(* IEC 61131-3 sources: ATCMcontrol_Engineering/src/COM/softing/fc/AddOns/Softing/4CPCTarget/Libs/ATCM_FLib, 23 files *)

(* ---- FA_SYNC_CLOSEFILE.st ---- *)
(*[[
    UserURL= "ATCM:FA_SYNC_CLOSEFILE.htm"
]]*)

(*
 *  ATCMControl FileAccess Function FA_SYNC_CLOSEFILE
 *  Purpose: Closes a file after read, write or getsize operation.
 *)
FUNCTION FA_SYNC_CLOSEFILE:BOOL     (* Return Value: error flag *)
VAR_INPUT
    EXEC        : BOOL;             (* start operation *)
END_VAR
VAR_IN_OUT
    FILE        : FA_SYNC_FILE;     (* file instance to operate on *)
END_VAR

inline
{
    ((COM.softing.fclib.flib.SyncFLib)%2).closeFile(%1)
}
END_FUNCTION

(* ---- FA_SYNC_CREATEDIRECTORY.st ---- *)
(*[[
    UserURL= "ATCM:FA_SYNC_CREATEDIRECTORY.htm"
]]*)

(*
 *  ATCMControl FileAccess Function FA_SYNC_CREATEDIRECTORY
 *  Purpose: Create a new directory.
 *)
FUNCTION FA_SYNC_CREATEDIRECTORY:BOOL   (* Return Value: error flag *)
VAR_INPUT
    EXEC        : BOOL;                 (* start operation *)
END_VAR
VAR_IN_OUT
    FILE        : FA_SYNC_FILE;         (* file instance to operate on *)
END_VAR

inline
{
    ((COM.softing.fclib.flib.SyncFLib)%2).createDir(%1)
}
END_FUNCTION

(* ---- FA_SYNC_DELETEFILE.st ---- *)
(*[[
    UserURL= "ATCM:FA_SYNC_DELETEFILE.htm"
]]*)

(*
 *  ATCMControl FileAccess Function FA_SYNC_DELETEFILE
 *  Purpose: Delete a file.
 *)
FUNCTION FA_SYNC_DELETEFILE:BOOL    (* Return Value: error flag *)
VAR_INPUT
    EXEC        : BOOL;             (* start operation *)
END_VAR
VAR_IN_OUT
    FILE        : FA_SYNC_FILE;     (* file instance to operate on *)
END_VAR

inline
{
    ((COM.softing.fclib.flib.SyncFLib)%2).deleteFile(%1)
}
END_FUNCTION

(* ---- FA_SYNC_EXISTSFILE.st ---- *)
(*[[
    UserURL= "ATCM:FA_SYNC_EXISTSFILE.htm"
]]*)

(*
 *  ATCMControl FileAccess Function FA_SYNC_EXISTSFILE
 *  Purpose: Determines whether a file exists.
 *)
FUNCTION FA_SYNC_EXISTSFILE:BOOL    (* Return Value: error flag *)
VAR_INPUT
    EXEC        : BOOL;             (* start operation *)
END_VAR
VAR_IN_OUT
    FILE        : FA_SYNC_FILE;     (* file instance to operate on *)
END_VAR
VAR_OUTPUT
    EXISTS      : BOOL;             (* TRUE if files exists, else FALSE *)
END_VAR

inline
{
    ((COM.softing.fclib.flib.SyncFLib)%2).existsFile(%1, %3)
}
END_FUNCTION

(* ---- FA_SYNC_GETSIZE.st ---- *)
(*[[
    UserURL= "ATCM:FA_SYNC_GETSIZE.htm"
]]*)

(*
 *  ATCMControl FileAccess Function FA_SYNC_GETSIZE
 *  Purpose: Retrieves the length in bytes of a file.
 *)
FUNCTION FA_SYNC_GETSIZE:BOOL       (* Return Value: error flag *)
VAR_INPUT
    EXEC        : BOOL;             (* start operation *)
END_VAR
VAR_IN_OUT
    FILE        : FA_SYNC_FILE;     (* file instance to operate on *)
END_VAR
VAR_OUTPUT
    SIZE        : LINT;             (* file size in bytes *)
END_VAR

inline
{
    ((COM.softing.fclib.flib.SyncFLib)%2).getSize(%1, %3)
}
END_FUNCTION

(* ---- FA_SYNC_OPENFILE.st ---- *)
(*[[
    UserURL= "ATCM:FA_SYNC_OPENFILE.htm"
]]*)

(*
 *  ATCMControl FileAccess Function FA_SYNC_OPENFILE
 *  Purpose: Opens a file for read, write or getsize operations.
 *)
FUNCTION FA_SYNC_OPENFILE:BOOL      (* Return Value: error flag *)
VAR_INPUT
    EXEC        : BOOL;             (* start operation *)
END_VAR
VAR_IN_OUT
    FILE        : FA_SYNC_FILE;     (* file instance to operate on *)
END_VAR

inline
{
    ((COM.softing.fclib.flib.SyncFLib)%2).createFile(%1)
}
END_FUNCTION

(* ---- FA_SYNC_READFILE.st ---- *)
(*[[
    UserURL= "ATCM:FA_SYNC_READFILE.htm"
]]*)

(*
 *  ATCMControl FileAccess Function FA_SYNC_READFILE
 *  Purpose: Reads data from a file.
 *)
FUNCTION FA_SYNC_READFILE:BOOL      (* Return Value: error flag *)
VAR_INPUT
    EXEC        : BOOL;             (* start operation *)
END_VAR
VAR_IN_OUT
    FILE        : FA_SYNC_FILE;     (* file instance to operate on *)
    LENGTH      : DINT;             (* bytes to read; return read bytes *)
END_VAR
VAR_OUTPUT
    DATA        : BYTE_STRING;      (* read data *)
END_VAR

inline
{
    ((COM.softing.fclib.flib.SyncFLib)%2).readFile(%1, %3, %4)
}
END_FUNCTION

(* ---- FA_SYNC_RENAMEFILE.st ---- *)
(*[[
    UserURL= "ATCM:FA_SYNC_RENAMEFILE.htm"
]]*)

(*
 *  ATCMControl FileAccess Function FA_SYNC_RENAMEFILE
 *  Purpose: Close file after read, write or getsize operation.
 *)
FUNCTION FA_SYNC_RENAMEFILE:BOOL    (* Return Value: error flag *)
VAR_INPUT
    EXEC        : BOOL;             (* start operation *)
    NEWNAME     : WSTRING;          (* new filename *)
END_VAR
VAR_IN_OUT
    FILE        : FA_SYNC_FILE;     (* file instance to operate on *)
END_VAR

inline
{
    ((COM.softing.fclib.flib.SyncFLib)%3).renameFile(%1, %2)
}
END_FUNCTION

(* ---- FA_SYNC_WRITEFILE.st ---- *)
(*[[
    UserURL= "ATCM:FA_SYNC_WRITEFILE.htm"
]]*)

(*
 *  ATCMControl FileAccess Function FA_SYNC_WRITEFILE
 *  Purpose: Writes data to a file.
 *)
FUNCTION FA_SYNC_WRITEFILE:BOOL     (* Return Value: error flag *)
VAR_INPUT
    EXEC        : BOOL;             (* start operation *)
    DATA        : BYTE_STRING;      (* data to write *)
END_VAR
VAR_IN_OUT
    FILE        : FA_SYNC_FILE;     (* file instance to operate on *)
END_VAR

inline
{
    ((COM.softing.fclib.flib.SyncFLib)%3).writeFile(%1, %2)
}
END_FUNCTION

(* ---- FA_ASYNC_CLOSEFILE.st ---- *)
(*[[
    UserURL= "ATCM:FA_ASYNC_CLOSEFILE.htm"
]]*)

(*
 *  ATCMControl FileAccess Functionblock FA_ASYNC_CLOSEFILE
 *  Purpose: Closes a file after read, write or getsize operation.
 *)
FUNCTION_BLOCK FA_ASYNC_CLOSEFILE
VAR_INPUT
    EXEC        : BOOL;             (* raising edge starts operation *)
END_VAR
VAR_IN_OUT
    FILE        : FA_ASYNC_FILE;    (* file instance to operate on *)
END_VAR
VAR_OUTPUT
    DONE        : BOOL;             (* operation finished *)
    ERROR       : BOOL;             (* error flag *)
    ERRCD       : DINT;             (* error code *)
    ERRTXT      : WSTRING;          (* error text *)
END_VAR

VAR
    rtrigExec   : R_TRIG;           (* execute *)
    token       : BOOL;             (* instance access token *)
    ireq        : BOOL;             (* execute request *)
END_VAR

rtrigExec(CLK := EXEC);
ireq := rtrigExec.Q;

NATIVE
    _done.putBool( ((COM.softing.fclib.flib.AsyncFLib)_file).closeFile(_exec.getBool(),
                        _ireq.getBool(),
                        _token,
                        this,
                        _error,
                        _errcd,
                        _errtxt) );
END_NATIVE;

END_FUNCTION_BLOCK

(* ---- FA_ASYNC_COPYFILE.st ---- *)
(*[[
    UserURL= "ATCM:FA_ASYNC_COPYFILE.htm"
]]*)

(*
 *  ATCMControl FileAccess Functionblock FA_ASYNC_COPYFILE
 *  Purpose: Copy a file.
 *)
FUNCTION_BLOCK FA_ASYNC_COPYFILE

VAR_INPUT
    EXEC        : BOOL;             (* raising edge starts operation *)
    DESTNAME    : WSTRING;          (* destination filename *)
    OVERWRITE   : BOOL := TRUE;     (* enable overwrite mode *)
END_VAR
VAR_IN_OUT
    FILE        : FA_ASYNC_FILE;    (* file instance to operate on *)
END_VAR
VAR_OUTPUT
    DONE        : BOOL;             (* operation finished *)
    ERROR       : BOOL;             (* error flag *)
    ERRCD       : DINT;             (* error code *)
    ERRTXT      : WSTRING;          (* error text *)
END_VAR

VAR
    rtrigExec   : R_TRIG;           (* execute *)
    token       : BOOL;             (* instance access token *)
    ireq        : BOOL;             (* execute request *)
END_VAR

rtrigExec(CLK := EXEC);
ireq := rtrigExec.Q;

NATIVE
    _done.putBool( ((COM.softing.fclib.flib.AsyncFLib)_file).copyFile(_exec.getBool(),
                        _ireq.getBool(),
                        _token,
                        this,
                        _destname.getString(),
                        _overwrite.getBool(),
                        _error,
                        _errcd,
                        _errtxt) );
END_NATIVE;

END_FUNCTION_BLOCK

(* ---- FA_ASYNC_CREATEDIRECTORY.st ---- *)
(*[[
    UserURL= "ATCM:FA_ASYNC_CREATEDIRECTORY.htm"
]]*)

(*
 *  ATCMControl FileAccess Functionblock FA_ASYNC_CREATEDIRECTORY
 *  Purpose: Create a new directory.
 *)
FUNCTION_BLOCK FA_ASYNC_CREATEDIRECTORY
VAR_INPUT
    EXEC        : BOOL;             (* raising edge starts operation *)
END_VAR
VAR_IN_OUT
    FILE        : FA_ASYNC_FILE;    (* file instance to operate on *)
END_VAR
VAR_OUTPUT
    DONE        : BOOL;             (* operation finished *)
    ERROR       : BOOL;             (* error flag *)
    ERRCD       : DINT;             (* error code *)
    ERRTXT      : WSTRING;          (* error text *)
END_VAR

VAR
    rtrigExec   : R_TRIG;           (* execute *)
    token       : BOOL;             (* instance access token *)
    ireq        : BOOL;             (* execute request *)
END_VAR

rtrigExec(CLK := EXEC);
ireq := rtrigExec.Q;

NATIVE
    _done.putBool( ((COM.softing.fclib.flib.AsyncFLib)_file).createDir(_exec.getBool(),
                        _ireq.getBool(),
                        _token,
                        this,
                        _error,
                        _errcd,
                        _errtxt) );
END_NATIVE;

END_FUNCTION_BLOCK

(* ---- FA_ASYNC_DELETEFILE.st ---- *)
(*[[
    UserURL= "ATCM:FA_ASYNC_DELETEFILE.htm"
]]*)

(*
 *  ATCMControl FileAccess Functionblock FA_ASYNC_DELETEFILE
 *  Purpose: Delete a file.
 *)
FUNCTION_BLOCK FA_ASYNC_DELETEFILE
VAR_INPUT
    EXEC        : BOOL;             (* raising edge starts operation *)
END_VAR
VAR_IN_OUT
    FILE        : FA_ASYNC_FILE;    (* file instance to operate on *)
END_VAR
VAR_OUTPUT
    DONE        : BOOL;             (* operation finished *)
    ERROR       : BOOL;             (* error flag *)
    ERRCD       : DINT;             (* error code *)
    ERRTXT      : WSTRING;          (* error text *)
END_VAR

VAR
    rtrigExec   : R_TRIG;           (* execute *)
    token       : BOOL;             (* instance access token *)
    ireq        : BOOL;             (* execute request *)
END_VAR

rtrigExec(CLK := EXEC);
ireq := rtrigExec.Q;

NATIVE
    _done.putBool( ((COM.softing.fclib.flib.AsyncFLib)_file).deleteFile(_exec.getBool(),
                        _ireq.getBool(),
                        _token,
                        this,
                        _error,
                        _errcd,
                        _errtxt) );
END_NATIVE;

END_FUNCTION_BLOCK

(* ---- FA_ASYNC_EXISTSFILE.st ---- *)
(*[[
    UserURL= "ATCM:FA_ASYNC_EXISTSFILE.htm"
]]*)

(*
 *  ATCMControl FileAccess Functionblock FA_ASYNC_EXISTSFILE
 *  Purpose: Determines whether a file exists.
 *)
FUNCTION_BLOCK FA_ASYNC_EXISTSFILE
VAR_INPUT
    EXEC        : BOOL;             (* raising edge starts operation *)
END_VAR
VAR_IN_OUT
    FILE        : FA_ASYNC_FILE;    (* file instance to operate on *)
END_VAR
VAR_OUTPUT
    EXISTS      : BOOL;             (* TRUE if files exists, else FALSE *)
    DONE        : BOOL;             (* operation finished *)
    ERROR       : BOOL;             (* error flag *)
    ERRCD       : DINT;             (* error code *)
    ERRTXT      : WSTRING;          (* error text *)
END_VAR

VAR
    rtrigExec   : R_TRIG;           (* execute *)
    token       : BOOL;             (* instance access token *)
    ireq        : BOOL;             (* execute request *)
END_VAR

rtrigExec(CLK := EXEC);
ireq := rtrigExec.Q;

NATIVE
    _done.putBool( ((COM.softing.fclib.flib.AsyncFLib)_file).existsFile(_exec.getBool(),
                        _ireq.getBool(),
                        _token,
                        this,
                        _exists,
                        _error,
                        _errcd,
                        _errtxt) );
END_NATIVE;

END_FUNCTION_BLOCK

(* ---- FA_ASYNC_GETSIZE.st ---- *)
(*[[
    UserURL= "ATCM:FA_ASYNC_GETSIZE.htm"
]]*)

(*
 *  ATCMControl FileAccess Functionblock FA_ASYNC_GETSIZE
 *  Purpose: Retrieves the length in bytes of a file.
 *)
FUNCTION_BLOCK FA_ASYNC_GETSIZE
VAR_INPUT
    EXEC        : BOOL;             (* raising edge starts operation *)
END_VAR
VAR_IN_OUT
    FILE        : FA_ASYNC_FILE;    (* file instance to operate on *)
END_VAR
VAR_OUTPUT
    SIZE        : LINT;             (* file size in bytes *)
    DONE        : BOOL;             (* operation finished *)
    ERROR       : BOOL;             (* error flag *)
    ERRCD       : DINT;             (* error code *)
    ERRTXT      : WSTRING;          (* error text *)
END_VAR

VAR
    rtrigExec   : R_TRIG;           (* execute *)
    token       : BOOL;             (* instance access token *)
    ireq        : BOOL;             (* execute request *)
END_VAR

rtrigExec(CLK := EXEC);
ireq := rtrigExec.Q;

NATIVE
    _done.putBool( ((COM.softing.fclib.flib.AsyncFLib)_file).getSize(_exec.getBool(),
                        _ireq.getBool(),
                        _token,
                        this,
                        (FcObject)_size,
                        _error,
                        _errcd,
                        _errtxt) );
END_NATIVE;

END_FUNCTION_BLOCK

(* ---- FA_ASYNC_OPENFILE.st ---- *)
(*[[
    UserURL= "ATCM:FA_ASYNC_OPENFILE.htm"
]]*)

(*
 *  ATCMControl FileAccess Functionblock FA_ASYNC_OPENFILE
 *  Purpose: Opens a file for read, write or getsize operations.
 *)
FUNCTION_BLOCK FA_ASYNC_OPENFILE
VAR_INPUT
    EXEC        : BOOL;             (* raising edge starts operation *)
END_VAR
VAR_IN_OUT
    FILE        : FA_ASYNC_FILE;    (* file instance to operate on *)
END_VAR
VAR_OUTPUT
    DONE        : BOOL;             (* operation finished *)
    ERROR       : BOOL;             (* error flag *)
    ERRCD       : DINT;             (* error code *)
    ERRTXT      : WSTRING;          (* error text *)
END_VAR

VAR
    rtrigExec   : R_TRIG;           (* execute *)
    token       : BOOL;             (* instance access token *)
    ireq        : BOOL;             (* execute request *)
END_VAR

rtrigExec(CLK := EXEC);
ireq := rtrigExec.Q;

NATIVE
    _done.putBool( ((COM.softing.fclib.flib.AsyncFLib)_file).createFile(_exec.getBool(),
                        _ireq.getBool(),
                        _token,
                        this,
                        _error,
                        _errcd,
                        _errtxt) );
END_NATIVE;

END_FUNCTION_BLOCK

(* ---- FA_ASYNC_READFILE.st ---- *)
(*[[
    UserURL= "ATCM:FA_ASYNC_READFILE.htm"
]]*)

(*
 *  ATCMControl FileAccess Functionblock FA_ASYNC_READFILE
 *  Purpose: Reads data from a file.
 *)

FUNCTION_BLOCK FA_ASYNC_READFILE
VAR_INPUT
    EXEC        : BOOL;             (* raising edge starts operation *)
END_VAR
VAR_IN_OUT
    FILE        : FA_ASYNC_FILE;    (* file instance to operate on *)
    LENGTH      : DINT;             (* bytes to read; return read bytes *)
END_VAR
VAR_OUTPUT
    DATA        : BYTE_STRING;      (* read data *)
    DONE        : BOOL;             (* operation finished *)
    ERROR       : BOOL;             (* error flag *)
    ERRCD       : DINT;             (* error code *)
    ERRTXT      : WSTRING;          (* error text *)
END_VAR

VAR
    rtrigExec   : R_TRIG;           (* execute *)
    token       : BOOL;             (* instance access token *)
    ireq        : BOOL;             (* execute request *)
END_VAR

rtrigExec(CLK := EXEC);
ireq := rtrigExec.Q;

NATIVE
    _done.putBool( ((COM.softing.fclib.flib.AsyncFLib)_file).readFile(_exec.getBool(),
                        _ireq.getBool(),
                        _token,
                        this,
                        (FcObject)_data,
                        _length,
                        _error,
                        _errcd,
                        _errtxt) );
END_NATIVE;

END_FUNCTION_BLOCK

(* ---- FA_ASYNC_RENAMEFILE.st ---- *)
(*[[
    UserURL= "ATCM:FA_ASYNC_RENAMEFILE.htm"
]]*)

(*
 *  ATCMControl FileAccess Functionblock FA_ASYNC_RENAMEFILE
 *  Purpose: Close file after read, write or getsize operation.
 *)
FUNCTION_BLOCK FA_ASYNC_RENAMEFILE
VAR_INPUT
    EXEC        : BOOL;             (* raising edge starts operation *)
    NEWNAME     : WSTRING;          (* new filename *)
END_VAR
VAR_IN_OUT
    FILE        : FA_ASYNC_FILE;    (* file instance to operate on *)
END_VAR
VAR_OUTPUT
    DONE        : BOOL;             (* operation finished *)
    ERROR       : BOOL;             (* error flag *)
    ERRCD       : DINT;             (* error code *)
    ERRTXT      : WSTRING;          (* error text *)
END_VAR

VAR
    rtrigExec   : R_TRIG;           (* execute *)
    token       : BOOL;             (* instance access token *)
    ireq        : BOOL;             (* execute request *)
END_VAR

rtrigExec(CLK := EXEC);
ireq := rtrigExec.Q;

NATIVE
    _done.putBool( ((COM.softing.fclib.flib.AsyncFLib)_file).renameFile(_exec.getBool(),
                        _ireq.getBool(),
                        _token,
                        this,
                        _newname.getString(),
                        _error,
                        _errcd,
                        _errtxt) );
END_NATIVE;

END_FUNCTION_BLOCK

(* ---- FA_ASYNC_WRITEFILE.st ---- *)
(*[[
    UserURL= "ATCM:FA_ASYNC_WRITEFILE.htm"
]]*)

(*
 *  ATCMControl FileAccess Functionblock FA_ASYNC_WRITEFILE
 *  Purpose: Writes data to a file.
 *)
FUNCTION_BLOCK FA_ASYNC_WRITEFILE
VAR_INPUT
    EXEC        : BOOL;             (* raising edge starts operation *)
    DATA        : BYTE_STRING;      (* data to write *)
END_VAR
VAR_IN_OUT
    FILE        : FA_ASYNC_FILE;    (* file instance to operate on *)
END_VAR
VAR_OUTPUT
    DONE        : BOOL;             (* operation finished *)
    ERROR       : BOOL;             (* error flag *)
    ERRCD       : DINT;             (* error code *)
    ERRTXT      : WSTRING;          (* error text *)
END_VAR

VAR
    rtrigExec   : R_TRIG;           (* execute *)
    token       : BOOL;             (* instance access token *)
    ireq        : BOOL;             (* execute request *)
END_VAR

rtrigExec(CLK := EXEC);
ireq := rtrigExec.Q;

NATIVE
    _done.putBool( ((COM.softing.fclib.flib.AsyncFLib)_file).writeFile(_exec.getBool(),
                        _ireq.getBool(),
                        _token,
                        this,
                        _data,
                        _error,
                        _errcd,
                        _errtxt) );
END_NATIVE;

END_FUNCTION_BLOCK

(* ---- FA_READFILE.st ---- *)
(*[[
    UserURL= "ATCM:FA_READFILE.htm"
]]*)

(*
 *  ATCMControl FileAccess Functionblock FA_READFILE
 *  Purpose: Reads data from a file.
 *)
FUNCTION_BLOCK FA_READFILE
VAR_INPUT
    EXEC        : BOOL;             (* raising edge starts operation *)
    FILENAME    : WSTRING;          (* filename *)
    TOUT        : TIME;             (* timeout for this operation *)
END_VAR
VAR_IN_OUT
    POSITION    : DINT;             (* start at position; returns last position *)
    LENGTH      : DINT;             (* bytes to read; returns read bytes *)
END_VAR
VAR_OUTPUT
    DATA        : BYTE_STRING;      (* read data *)
    DONE        : BOOL;             (* operation finished *)
    ERROR       : BOOL;             (* error flag *)
    ERRCD       : DINT;             (* error code *)
    ERRTXT      : WSTRING;          (* error text *)
END_VAR

VAR
    file        : FA_ASYNC_FILE;
    aopen       : FA_ASYNC_OPENFILE;
    aread       : FA_ASYNC_READFILE;
    aclose      : FA_ASYNC_CLOSEFILE;
    rtDone      : R_TRIG;
    rtInit      : R_TRIG;
    rtRead      : R_TRIG;
    rtError     : R_TRIG;
    bstrData    : BYTE_STRING;
END_VAR

(* init structure *)
file.FILENAME := FILENAME;
file.MODE := CFA_READ;
(* file.TEXTMODE is default: FALSE *)
file.TOUT := TOUT;

(* delete output *)
IF NOT EXEC THEN
    DONE := FALSE;
    ERROR := FALSE;
    ERRCD := 0;
    ERRTXT := "";
    BYTE_STRING_INIT(DATA, "");
    file.ISERROR := FALSE;
END_IF;

(* open file *)
aopen(EXEC := EXEC, FILE := file);

(* init read file *)
rtInit(CLK := aopen.DONE);
IF rtInit.Q THEN
    (* init *)
    file.POSITION := POSITION;
END_IF;
aread(EXEC := aopen.DONE AND NOT aopen.ERROR, FILE := file, LENGTH := LENGTH);
(* read file done *)
rtRead(CLK := aread.DONE);
IF rtRead.Q THEN
    bstrData := aread.DATA;
END_IF;

(* close file *)
aclose(EXEC := aread.DONE AND NOT aread.ERROR, FILE := file);

(* init output vars *)
rtDone(CLK := aclose.DONE);
IF rtDone.Q THEN
    DONE        := TRUE;
    DATA        := bstrData;
    POSITION    := file.POSITION;
END_IF;

(* init error vars *)
rtError(CLK := file.ISERROR);
IF rtError.Q THEN
    DONE        := TRUE;
    BYTE_STRING_INIT(DATA, "");
    ERROR       := file.ISERROR;
    ERRCD       := file.LSTERRCD;
    ERRTXT      := file.LSTERRTXT;
END_IF;

END_FUNCTION_BLOCK

(* ---- FA_READLINE.st ---- *)
(*[[
    UserURL= "ATCM:FA_READLINE.htm"
]]*)

(*
 *  ATCMControl FileAccess Functionblock FA_READLINE
 *  Purpose: Reads data from a file.
 *)
FUNCTION_BLOCK FA_READLINE
VAR_INPUT
    EXEC        : BOOL;             (* raising edge starts operation *)
    FILENAME    : WSTRING;          (* filename *)
    TOUT        : TIME;             (* timeout for this operation *)
END_VAR
VAR_IN_OUT
    POSITION    : DINT;             (* start at position; returns last position *)
END_VAR
VAR_OUTPUT
    DATA        : WSTRING;          (* read data *)
    DONE        : BOOL;             (* operation finished *)
    ERROR       : BOOL;             (* error flag *)
    ERRCD       : DINT;             (* error code *)
    ERRTXT      : WSTRING;          (* error text *)
END_VAR

VAR
    file        : FA_ASYNC_FILE;
    aopen       : FA_ASYNC_OPENFILE;
    aread       : FA_ASYNC_READFILE;
    aclose      : FA_ASYNC_CLOSEFILE;
    length      : DINT;
    rtDone      : R_TRIG;
    rtInit      : R_TRIG;
    rtRead      : R_TRIG;
    rtError     : R_TRIG;
    pos         : DINT;
    bstrData    : BYTE_STRING;
END_VAR

(* init structure *)
file.FILENAME := FILENAME;
file.MODE := CFA_READ;
file.TEXTMODE := TRUE;
file.TOUT := TOUT;
length := CFA_EOL;

(* delete output *)
IF NOT EXEC THEN
    DONE := FALSE;
    ERROR := FALSE;
    ERRCD := 0;
    ERRTXT := "";
    DATA := "";
    file.ISERROR := FALSE;
END_IF;

(* open file *)
aopen(EXEC := EXEC, FILE := file);

(* init read file *)
rtInit(CLK := aopen.DONE);
IF rtInit.Q THEN
    (* init *)
    file.POSITION := POSITION;
END_IF;
aread(EXEC := aopen.DONE AND NOT aopen.ERROR, FILE := file, LENGTH := length);
(* read file done *)
rtRead(CLK := aread.DONE);
IF rtRead.Q THEN
    bstrData := aread.DATA;
END_IF;

(* close file *)
aclose(EXEC := aread.DONE AND NOT aread.ERROR, FILE := file);

(* init output vars *)
rtDone(CLK := aclose.DONE);
IF rtDone.Q THEN
    DONE        := TRUE;
    (* convert WString to BYTE_STRING *)
    pos := 0;
    DATA        := COPY_WSTRING_FROM_BYTE_STRING(bstrdata.SIZE, pos, bstrdata);
    POSITION    := file.POSITION;
END_IF;

(* init error vars *)
rtError(CLK := file.ISERROR);
IF rtError.Q THEN
    DONE        := TRUE;
    DATA        := "";
    ERROR       := file.ISERROR;
    ERRCD       := file.LSTERRCD;
    ERRTXT      := file.LSTERRTXT;
END_IF;

END_FUNCTION_BLOCK

(* ---- FA_WRITEFILE.st ---- *)
(*[[
    UserURL= "ATCM:FA_WRITEFILE.htm"
]]*)

(*
 *  ATCMControl FileAccess Functionblock FA_WRITEFILE
 *  Purpose: Writes data to a file.
 *)
FUNCTION_BLOCK FA_WRITEFILE
VAR_INPUT
    EXEC        : BOOL;             (* raising edge starts operation *)
    FILENAME    : WSTRING;          (* filename *)
    TOUT        : TIME;             (* timeout for this operation *)
    DATA        : BYTE_STRING;      (* data to write *)
END_VAR
VAR_IN_OUT
    POSITION    : DINT;             (* start at position; returns last position *)
END_VAR
VAR_OUTPUT
    DONE        : BOOL;             (* operation finished *)
    ERROR       : BOOL;             (* error flag *)
    ERRCD       : DINT;             (* error code *)
    ERRTXT      : WSTRING;          (* error text *)
END_VAR

VAR
    file        : FA_ASYNC_FILE;
    aopen       : FA_ASYNC_OPENFILE;
    awrite      : FA_ASYNC_WRITEFILE;
    aclose      : FA_ASYNC_CLOSEFILE;
    rtWrite     : R_TRIG;
    rtDone      : R_TRIG;
    rtError     : R_TRIG;
    posPtr      : DINT;
END_VAR

(* init structure *)
file.FILENAME := FILENAME;
file.MODE := CFA_READ_WRITE;
(* file.TEXTMODE is default: FALSE *)
file.TOUT := TOUT;

(* delete output *)
IF NOT EXEC THEN
    DONE := FALSE;
    ERROR := FALSE;
    ERRCD := 0;
    ERRTXT := "";
    file.ISERROR := FALSE;
END_IF;

(* open file *)
aopen(EXEC := EXEC, FILE := file);

(* read file *)
file.POSITION := POSITION;
awrite(EXEC := aopen.DONE AND NOT aopen.ERROR, FILE := file, DATA := DATA);
(* write file done *)
rtWrite(CLK := awrite.DONE);
IF rtWrite.Q THEN
    posPtr := file.POSITION;
END_IF;

(* close file *)
aclose(EXEC := awrite.DONE, FILE := file);

(* init output vars *)
rtDone(CLK := aclose.DONE);
IF rtDone.Q THEN
    DONE        := TRUE;
    POSITION    := posPtr;
END_IF;

(* init error vars *)
rtError(CLK := file.ISERROR);
IF rtError.Q THEN
    DONE        := TRUE;
    ERROR       := file.ISERROR;
    ERRCD       := file.LSTERRCD;
    ERRTXT      := file.LSTERRTXT;
END_IF;

END_FUNCTION_BLOCK

(* ---- FA_WRITELINE.st ---- *)
(*[[
    UserURL= "ATCM:FA_WRITELINE.htm"
]]*)

(*
 *  ATCMControl FileAccess Functionblock FA_WRITELINE
 *  Purpose: Writes data to a file.
 *)
FUNCTION_BLOCK FA_WRITELINE
VAR_INPUT
    EXEC        : BOOL;             (* raising edge starts operation *)
    FILENAME    : WSTRING;          (* filename *)
    TOUT        : TIME;             (* timeout for this operation *)
    DATA        : WSTRING;          (* data to write *)
END_VAR
VAR_IN_OUT
    POSITION    : DINT;             (* start at position; returns last position *)
END_VAR
VAR_OUTPUT
    DONE        : BOOL;             (* operation finished *)
    ERROR       : BOOL;             (* error flag *)
    ERRCD       : DINT;             (* error code *)
    ERRTXT      : WSTRING;          (* error text *)
END_VAR

VAR
    file        : FA_ASYNC_FILE;
    aopen       : FA_ASYNC_OPENFILE;
    awrite      : FA_ASYNC_WRITEFILE;
    aclose      : FA_ASYNC_CLOSEFILE;
    length      : DINT;
    ldata       : WSTRING;
    bstrData    : BYTE_STRING;
    rtWrite     : R_TRIG;
    rtDone      : R_TRIG;
    rtInit      : R_TRIG;
    rtError     : R_TRIG;
    posStr      : DINT := 0;
    posPtr      : DINT;
END_VAR

(* init structure *)
file.FILENAME := FILENAME;
file.MODE := CFA_READ_WRITE;
file.TEXTMODE := TRUE;
file.TOUT := TOUT;

(* delete output *)
IF NOT EXEC THEN
    DONE := FALSE;
    ERROR := FALSE;
    ERRCD := 0;
    ERRTXT := "";
    file.ISERROR := FALSE;
END_IF;

(* open file *)
aopen(EXEC := EXEC, FILE := file);

(* init write file *)
rtInit(CLK := aopen.DONE);
IF rtInit.Q THEN
    (* init *)
    file.POSITION := POSITION;
    (* convert WString to BYTE_STRING *)
    posStr := 0;
    COPY_WSTRING_TO_BYTE_STRING(CONCAT(DATA, "$n"), posStr, bstrData);
    bstrData.size := posStr;
END_IF;
(* write into file *)
awrite(EXEC := aopen.DONE AND NOT aopen.ERROR, FILE := file, DATA := bstrData);
(* write file done *)
rtWrite(CLK := awrite.DONE);
IF rtWrite.Q THEN
    posPtr := file.POSITION;
END_IF;

(* close file *)
aclose(EXEC := awrite.DONE, FILE := file);

(* init output vars *)
rtDone(CLK := aclose.DONE);
IF rtDone.Q THEN
    DONE        := TRUE;
    POSITION    := posPtr;
END_IF;

(* init error vars *)
rtError(CLK := file.ISERROR);
IF rtError.Q THEN
    DONE        := TRUE;
    ERROR       := file.ISERROR;
    ERRCD       := file.LSTERRCD;
    ERRTXT      := file.LSTERRTXT;
END_IF;

END_FUNCTION_BLOCK
